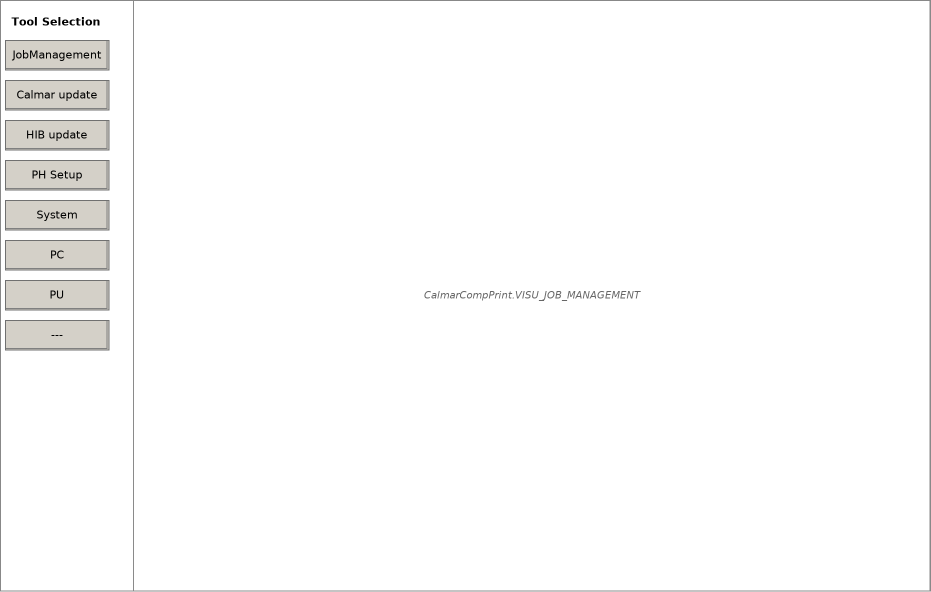
VISUALIZATION VISU_SERVICE  // 931x592
    Button (5,80 104x30), "Calmar update", colour toggle: PRG_PRINT.nServiceVisuFrameIndex = 1
        OnMouseClick: execute { PRG_PRINT.nServiceVisuFrameIndex := 1; }
    Button (5,40 104x30), "JobManagement", colour toggle: PRG_PRINT.nServiceVisuFrameIndex = 0
        OnMouseClick: execute { PRG_PRINT.nServiceVisuFrameIndex := 0; }
    Button (5,120 104x30), "HIB update", colour toggle: PRG_PRINT.nServiceVisuFrameIndex = 2
        OnMouseClick: execute { PRG_PRINT.nServiceVisuFrameIndex := 2; }
    Button (5,160 104x30), "PH Setup", colour toggle: PRG_PRINT.nServiceVisuFrameIndex = 3
        OnMouseClick: execute { PRG_PRINT.nServiceVisuFrameIndex := 3; }
    Button (5,200 104x30), "System", colour toggle: PRG_PRINT.nServiceVisuFrameIndex = 4
        OnMouseClick: execute { PRG_PRINT.nServiceVisuFrameIndex := 4; }
    Rectangle (4,7 104x30), "Tool Selection"
    Frame (133,-1 798x592), frame switch variable: PRG_PRINT.nServiceVisuFrameIndex
        shows CalmarCompPrint.VISU_JOB_MANAGEMENT(m_Fb_JobManagement := PRG_PRINT.fbPrgPrintTest.fb_JobManagement)
        shows CalmarCompPrint.VISU_SETUP_CALMAR(m_fb_calmar_upd := PRG_PRINT.fb_fwhw_update)
        shows CalmarCompPrint.VISU_SETUP_HIB(m_visu_fb := PRG_PRINT.fb_hib_rup)
        shows CalmarCompPrint.VISU_SETUP_PH(m_Inst_fb_wave := PRG_PRINT.fb_fdl_waveform, m_Inst_fb_mask := PRG_PRINT.fb_fdl_mask)
        shows CalmarCompSystem.VISU_SYSTEM()
        shows CalmarCompPrint.VISU_PC(m_visu_fb := PRG_PRINT.fb_visu_pc)
        shows CalmarCompPrint.VISU_PU(m_visu_fb := PRG_PRINT.fb_visu_pu)
        p2546873765: PRG_PRINT.fb_fdl_imgmap
        p2204176931: PRG_PRINT.fb_visu_pu
    Button (5,240 104x30), "PC", colour toggle: PRG_PRINT.nServiceVisuFrameIndex = 5
        OnMouseClick: execute { PRG_PRINT.nServiceVisuFrameIndex := 5; }
    Button (5,280 104x30), "PU", colour toggle: PRG_PRINT.nServiceVisuFrameIndex = 6
        OnMouseClick: execute { PRG_PRINT.nServiceVisuFrameIndex := 6; }
    Button (5,320 104x30), "---", colour toggle: PRG_PRINT.nServiceVisuFrameIndex = 7
        OnMouseClick: execute { PRG_PRINT.nServiceVisuFrameIndex := 7; }
END_VISUALIZATION

(* stored: Version 1.1.0.1, ProductVersion 3.1.4024.4
   Visu VISU_SERVICE: Id {909ae22e-b5e2-4752-9d7c-ebeb0086d62f} *)
